// TIA Portal V18 export
FUNCTION_BLOCK "CentralShifter"   // FB10, LAD
{ S7_Optimized_Access := 'TRUE' }
// stored: MemoryReserve 100, SetENOAutomatically false
   VAR
      MC_POWER_CS_PP { S7_SetPoint := 'True'} : MC_POWER;
      MC_POWER_CS_PL { S7_SetPoint := 'True'} : MC_POWER;
      MC_POWER_CS_TP { S7_SetPoint := 'True'} : MC_POWER;
      MC_POWER_CS_TL { S7_SetPoint := 'True'} : MC_POWER;
      MC_POWER_CS_Virtual { S7_SetPoint := 'True'} : MC_POWER;
      MC_RESET_CS_PP { S7_SetPoint := 'True'} : MC_RESET;
      MC_RESET_CS_PL { S7_SetPoint := 'True'} : MC_RESET;
      MC_RESET_CS_TP { S7_SetPoint := 'True'} : MC_RESET;
      MC_RESET_CS_TL { S7_SetPoint := 'True'} : MC_RESET;
      MC_GEARIN_CS_PP { S7_SetPoint := 'True'} : MC_GEARIN;
      MC_GEARIN_CS_PL { S7_SetPoint := 'True'} : MC_GEARIN;
      MC_GEARIN_CS_TP { S7_SetPoint := 'True'} : MC_GEARIN;
      MC_GEARIN_CS_TL { S7_SetPoint := 'True'} : MC_GEARIN;
      MC_HOME_CS_PP { S7_SetPoint := 'True'} : MC_HOME;
      MC_HOME_CS_PL { S7_SetPoint := 'True'} : MC_HOME;
      MC_HOME_CS_TP { S7_SetPoint := 'True'} : MC_HOME;
      MC_HOME_CS_TL { S7_SetPoint := 'True'} : MC_HOME;
      MC_RESET_CS_Virtual { S7_SetPoint := 'True'} : MC_RESET;
      MC_MOVEJOG_CS_PL { S7_SetPoint := 'True'} : MC_MOVEJOG;
      MC_HOME_CS_Virtual { S7_SetPoint := 'True'} : MC_HOME;
      MC_MOVEJOG_CS_PP { S7_SetPoint := 'True'} : MC_MOVEJOG;
      MC_MOVEJOG_CS_TL { S7_SetPoint := 'True'} : MC_MOVEJOG;
      MC_MOVEJOG_CS_TP { S7_SetPoint := 'True'} : MC_MOVEJOG;
      MC_MOVEJOG_CS_Virtual { S7_SetPoint := 'True'} : MC_MOVEJOG;
      MC_MOVERELATIVE_CS_Virtual { S7_SetPoint := 'True'} : MC_MOVERELATIVE;
      MC_MOVEABSOLUTE_CS_Virtual { S7_SetPoint := 'True'} : MC_MOVEABSOLUTE;
      Homeing_Status { S7_SetPoint := 'True'} : Int;
      Jog_Backward_Home : Bool;
      Jog_Forward_Home : Bool;
      Jog_Velocity : Int;
   END_VAR
BEGIN

REGION Network 1
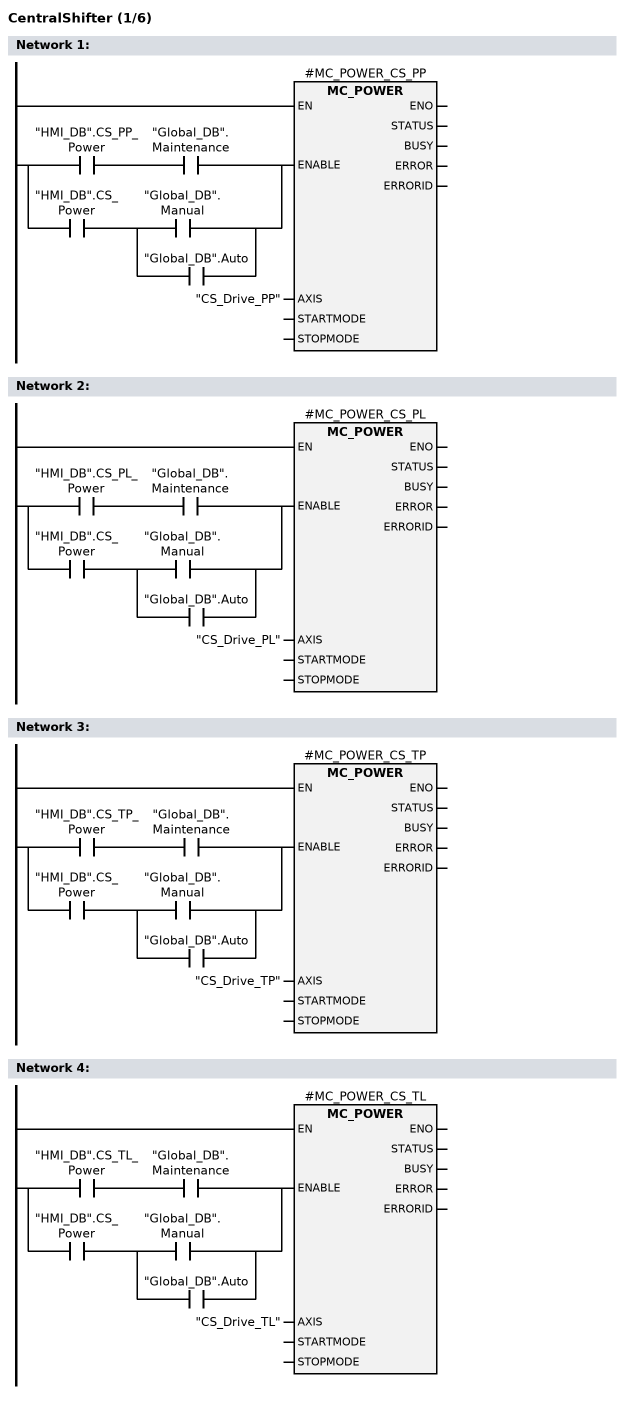
   RUNG wire#powerrail
      #MC_POWER_CS_PP.MC_POWER(Enable := wire#w2, Axis := "CS_Drive_PP", StartMode :=, StopMode :=, Status =>, Busy =>, Error =>, ErrorId =>)
   END_RUNG
   RUNG wire#powerrail
      Contact( "HMI_DB".CS_PP_Power )
      Contact( "Global_DB".Maintenance )
   END_RUNG wire#w2
   RUNG wire#powerrail
      Contact( "HMI_DB".CS_Power )
      wire#w1
      Contact( "Global_DB".Manual )
   END_RUNG wire#w2
   RUNG wire#w1
      Contact( "Global_DB".Auto )
   END_RUNG wire#w2
   // the same network as SCL:
   #MC_POWER_CS_PP(Enable := ("HMI_DB".CS_PP_Power AND "Global_DB".Maintenance) OR ("HMI_DB".CS_Power AND ("Global_DB".Manual OR "Global_DB".Auto)),   // MC_POWER
                   Axis := "CS_Drive_PP");
END_REGION

REGION Network 2
   RUNG wire#powerrail
      #MC_POWER_CS_PL.MC_POWER(Enable := wire#w2, Axis := "CS_Drive_PL", StartMode :=, StopMode :=, Status =>, Busy =>, Error =>, ErrorId =>)
   END_RUNG
   RUNG wire#powerrail
      Contact( "HMI_DB".CS_PL_Power )
      Contact( "Global_DB".Maintenance )
   END_RUNG wire#w2
   RUNG wire#powerrail
      Contact( "HMI_DB".CS_Power )
      wire#w1
      Contact( "Global_DB".Manual )
   END_RUNG wire#w2
   RUNG wire#w1
      Contact( "Global_DB".Auto )
   END_RUNG wire#w2
   // the same network as SCL:
   #MC_POWER_CS_PL(Enable := ("HMI_DB".CS_PL_Power AND "Global_DB".Maintenance) OR ("HMI_DB".CS_Power AND ("Global_DB".Manual OR "Global_DB".Auto)),   // MC_POWER
                   Axis := "CS_Drive_PL");
END_REGION

REGION Network 3
   RUNG wire#powerrail
      #MC_POWER_CS_TP.MC_POWER(Enable := wire#w2, Axis := "CS_Drive_TP", StartMode :=, StopMode :=, Status =>, Busy =>, Error =>, ErrorId =>)
   END_RUNG
   RUNG wire#powerrail
      Contact( "HMI_DB".CS_TP_Power )
      Contact( "Global_DB".Maintenance )
   END_RUNG wire#w2
   RUNG wire#powerrail
      Contact( "HMI_DB".CS_Power )
      wire#w1
      Contact( "Global_DB".Manual )
   END_RUNG wire#w2
   RUNG wire#w1
      Contact( "Global_DB".Auto )
   END_RUNG wire#w2
   // the same network as SCL:
   #MC_POWER_CS_TP(Enable := ("HMI_DB".CS_TP_Power AND "Global_DB".Maintenance) OR ("HMI_DB".CS_Power AND ("Global_DB".Manual OR "Global_DB".Auto)),   // MC_POWER
                   Axis := "CS_Drive_TP");
END_REGION

REGION Network 4
   RUNG wire#powerrail
      #MC_POWER_CS_TL.MC_POWER(Enable := wire#w2, Axis := "CS_Drive_TL", StartMode :=, StopMode :=, Status =>, Busy =>, Error =>, ErrorId =>)
   END_RUNG
   RUNG wire#powerrail
      Contact( "HMI_DB".CS_TL_Power )
      Contact( "Global_DB".Maintenance )
   END_RUNG wire#w2
   RUNG wire#powerrail
      Contact( "HMI_DB".CS_Power )
      wire#w1
      Contact( "Global_DB".Manual )
   END_RUNG wire#w2
   RUNG wire#w1
      Contact( "Global_DB".Auto )
   END_RUNG wire#w2
   // the same network as SCL:
   #MC_POWER_CS_TL(Enable := ("HMI_DB".CS_TL_Power AND "Global_DB".Maintenance) OR ("HMI_DB".CS_Power AND ("Global_DB".Manual OR "Global_DB".Auto)),   // MC_POWER
                   Axis := "CS_Drive_TL");
END_REGION

REGION Network 5
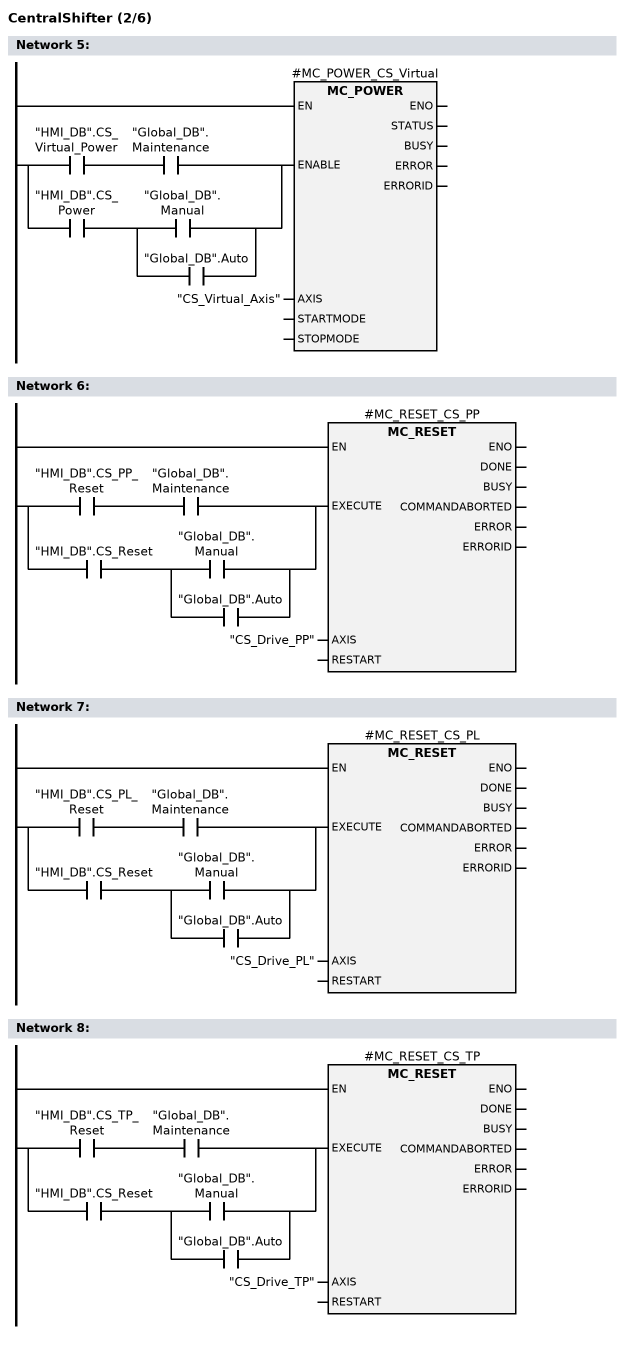
   RUNG wire#powerrail
      #MC_POWER_CS_Virtual.MC_POWER(Enable := wire#w2, Axis := "CS_Virtual_Axis", StartMode :=, StopMode :=, Status =>, Busy =>, Error =>, ErrorId =>)
   END_RUNG
   RUNG wire#powerrail
      Contact( "HMI_DB".CS_Virtual_Power )
      Contact( "Global_DB".Maintenance )
   END_RUNG wire#w2
   RUNG wire#powerrail
      Contact( "HMI_DB".CS_Power )
      wire#w1
      Contact( "Global_DB".Manual )
   END_RUNG wire#w2
   RUNG wire#w1
      Contact( "Global_DB".Auto )
   END_RUNG wire#w2
   // the same network as SCL:
   #MC_POWER_CS_Virtual(Enable := ("HMI_DB".CS_Virtual_Power AND "Global_DB".Maintenance) OR ("HMI_DB".CS_Power AND ("Global_DB".Manual OR "Global_DB".Auto)),   // MC_POWER
                        Axis := "CS_Virtual_Axis");
END_REGION

REGION Network 6
   RUNG wire#powerrail
      #MC_RESET_CS_PP.MC_RESET(Execute := wire#w2, Axis := "CS_Drive_PP", Restart :=, Done =>, Busy =>, CommandAborted =>, Error =>, ErrorId =>)
   END_RUNG
   RUNG wire#powerrail
      Contact( "HMI_DB".CS_PP_Reset )
      Contact( "Global_DB".Maintenance )
   END_RUNG wire#w2
   RUNG wire#powerrail
      Contact( "HMI_DB".CS_Reset )
      wire#w1
      Contact( "Global_DB".Manual )
   END_RUNG wire#w2
   RUNG wire#w1
      Contact( "Global_DB".Auto )
   END_RUNG wire#w2
   // the same network as SCL:
   #MC_RESET_CS_PP(Execute := ("HMI_DB".CS_PP_Reset AND "Global_DB".Maintenance) OR ("HMI_DB".CS_Reset AND ("Global_DB".Manual OR "Global_DB".Auto)),   // MC_RESET
                   Axis := "CS_Drive_PP");
END_REGION

REGION Network 7
   RUNG wire#powerrail
      #MC_RESET_CS_PL.MC_RESET(Execute := wire#w2, Axis := "CS_Drive_PL", Restart :=, Done =>, Busy =>, CommandAborted =>, Error =>, ErrorId =>)
   END_RUNG
   RUNG wire#powerrail
      Contact( "HMI_DB".CS_PL_Reset )
      Contact( "Global_DB".Maintenance )
   END_RUNG wire#w2
   RUNG wire#powerrail
      Contact( "HMI_DB".CS_Reset )
      wire#w1
      Contact( "Global_DB".Manual )
   END_RUNG wire#w2
   RUNG wire#w1
      Contact( "Global_DB".Auto )
   END_RUNG wire#w2
   // the same network as SCL:
   #MC_RESET_CS_PL(Execute := ("HMI_DB".CS_PL_Reset AND "Global_DB".Maintenance) OR ("HMI_DB".CS_Reset AND ("Global_DB".Manual OR "Global_DB".Auto)),   // MC_RESET
                   Axis := "CS_Drive_PL");
END_REGION

REGION Network 8
   RUNG wire#powerrail
      #MC_RESET_CS_TP.MC_RESET(Execute := wire#w2, Axis := "CS_Drive_TP", Restart :=, Done =>, Busy =>, CommandAborted =>, Error =>, ErrorId =>)
   END_RUNG
   RUNG wire#powerrail
      Contact( "HMI_DB".CS_TP_Reset )
      Contact( "Global_DB".Maintenance )
   END_RUNG wire#w2
   RUNG wire#powerrail
      Contact( "HMI_DB".CS_Reset )
      wire#w1
      Contact( "Global_DB".Manual )
   END_RUNG wire#w2
   RUNG wire#w1
      Contact( "Global_DB".Auto )
   END_RUNG wire#w2
   // the same network as SCL:
   #MC_RESET_CS_TP(Execute := ("HMI_DB".CS_TP_Reset AND "Global_DB".Maintenance) OR ("HMI_DB".CS_Reset AND ("Global_DB".Manual OR "Global_DB".Auto)),   // MC_RESET
                   Axis := "CS_Drive_TP");
END_REGION

REGION Network 9
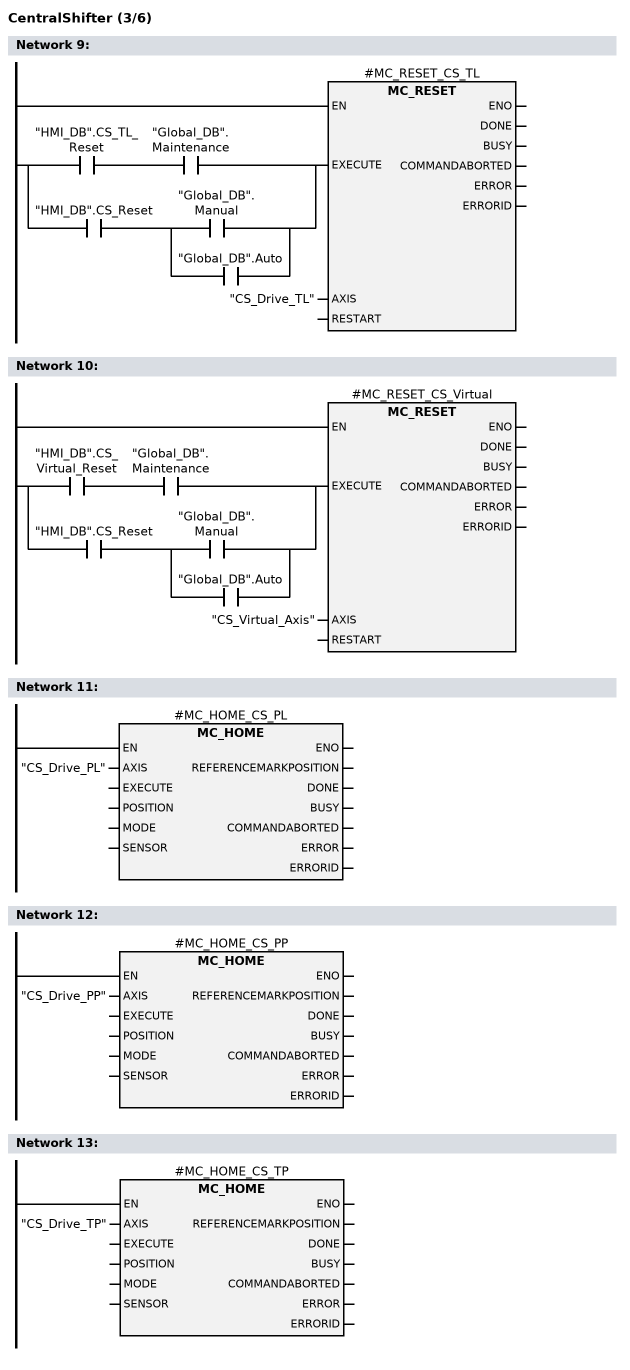
   RUNG wire#powerrail
      #MC_RESET_CS_TL.MC_RESET(Execute := wire#w2, Axis := "CS_Drive_TL", Restart :=, Done =>, Busy =>, CommandAborted =>, Error =>, ErrorId =>)
   END_RUNG
   RUNG wire#powerrail
      Contact( "HMI_DB".CS_TL_Reset )
      Contact( "Global_DB".Maintenance )
   END_RUNG wire#w2
   RUNG wire#powerrail
      Contact( "HMI_DB".CS_Reset )
      wire#w1
      Contact( "Global_DB".Manual )
   END_RUNG wire#w2
   RUNG wire#w1
      Contact( "Global_DB".Auto )
   END_RUNG wire#w2
   // the same network as SCL:
   #MC_RESET_CS_TL(Execute := ("HMI_DB".CS_TL_Reset AND "Global_DB".Maintenance) OR ("HMI_DB".CS_Reset AND ("Global_DB".Manual OR "Global_DB".Auto)),   // MC_RESET
                   Axis := "CS_Drive_TL");
END_REGION

REGION Network 10
   RUNG wire#powerrail
      #MC_RESET_CS_Virtual.MC_RESET(Execute := wire#w2, Axis := "CS_Virtual_Axis", Restart :=, Done =>, Busy =>, CommandAborted =>, Error =>, ErrorId =>)
   END_RUNG
   RUNG wire#powerrail
      Contact( "HMI_DB".CS_Virtual_Reset )
      Contact( "Global_DB".Maintenance )
   END_RUNG wire#w2
   RUNG wire#powerrail
      Contact( "HMI_DB".CS_Reset )
      wire#w1
      Contact( "Global_DB".Manual )
   END_RUNG wire#w2
   RUNG wire#w1
      Contact( "Global_DB".Auto )
   END_RUNG wire#w2
   // the same network as SCL:
   #MC_RESET_CS_Virtual(Execute := ("HMI_DB".CS_Virtual_Reset AND "Global_DB".Maintenance) OR ("HMI_DB".CS_Reset AND ("Global_DB".Manual OR "Global_DB".Auto)),   // MC_RESET
                        Axis := "CS_Virtual_Axis");
END_REGION

REGION Network 11
   RUNG wire#powerrail
      #MC_HOME_CS_PL.MC_HOME(Axis := "CS_Drive_PL", Execute :=, Position :=, Mode :=, Sensor :=, ReferenceMarkPosition =>, Done =>, Busy =>, CommandAborted =>, Error =>, ErrorId =>)
   END_RUNG
   // the same network as SCL:
   #MC_HOME_CS_PL(Axis := "CS_Drive_PL");   // MC_HOME
END_REGION

REGION Network 12
   RUNG wire#powerrail
      #MC_HOME_CS_PP.MC_HOME(Axis := "CS_Drive_PP", Execute :=, Position :=, Mode :=, Sensor :=, ReferenceMarkPosition =>, Done =>, Busy =>, CommandAborted =>, Error =>, ErrorId =>)
   END_RUNG
   // the same network as SCL:
   #MC_HOME_CS_PP(Axis := "CS_Drive_PP");   // MC_HOME
END_REGION

REGION Network 13
   RUNG wire#powerrail
      #MC_HOME_CS_TP.MC_HOME(Axis := "CS_Drive_TP", Execute :=, Position :=, Mode :=, Sensor :=, ReferenceMarkPosition =>, Done =>, Busy =>, CommandAborted =>, Error =>, ErrorId =>)
   END_RUNG
   // the same network as SCL:
   #MC_HOME_CS_TP(Axis := "CS_Drive_TP");   // MC_HOME
END_REGION

REGION Network 14
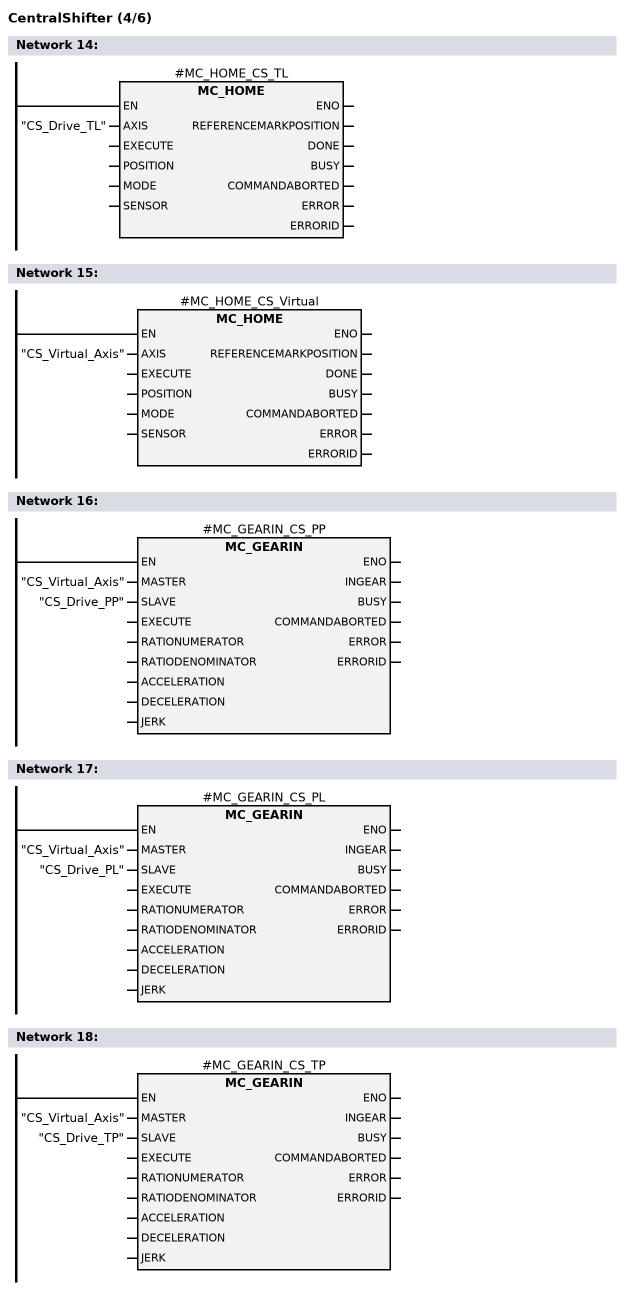
   RUNG wire#powerrail
      #MC_HOME_CS_TL.MC_HOME(Axis := "CS_Drive_TL", Execute :=, Position :=, Mode :=, Sensor :=, ReferenceMarkPosition =>, Done =>, Busy =>, CommandAborted =>, Error =>, ErrorId =>)
   END_RUNG
   // the same network as SCL:
   #MC_HOME_CS_TL(Axis := "CS_Drive_TL");   // MC_HOME
END_REGION

REGION Network 15
   RUNG wire#powerrail
      #MC_HOME_CS_Virtual.MC_HOME(Axis := "CS_Virtual_Axis", Execute :=, Position :=, Mode :=, Sensor :=, ReferenceMarkPosition =>, Done =>, Busy =>, CommandAborted =>, Error =>, ErrorId =>)
   END_RUNG
   // the same network as SCL:
   #MC_HOME_CS_Virtual(Axis := "CS_Virtual_Axis");   // MC_HOME
END_REGION

REGION Network 16
   RUNG wire#powerrail
      #MC_GEARIN_CS_PP.MC_GEARIN(Master := "CS_Virtual_Axis", Slave := "CS_Drive_PP", Execute :=, RatioNumerator :=, RatioDenominator :=, Acceleration :=, Deceleration :=, Jerk :=, InGear =>, Busy =>, CommandAborted =>, Error =>, ErrorId =>)
   END_RUNG
   // the same network as SCL:
   #MC_GEARIN_CS_PP(Master := "CS_Virtual_Axis", Slave := "CS_Drive_PP");   // MC_GEARIN
END_REGION

REGION Network 17
   RUNG wire#powerrail
      #MC_GEARIN_CS_PL.MC_GEARIN(Master := "CS_Virtual_Axis", Slave := "CS_Drive_PL", Execute :=, RatioNumerator :=, RatioDenominator :=, Acceleration :=, Deceleration :=, Jerk :=, InGear =>, Busy =>, CommandAborted =>, Error =>, ErrorId =>)
   END_RUNG
   // the same network as SCL:
   #MC_GEARIN_CS_PL(Master := "CS_Virtual_Axis", Slave := "CS_Drive_PL");   // MC_GEARIN
END_REGION

REGION Network 18
   RUNG wire#powerrail
      #MC_GEARIN_CS_TP.MC_GEARIN(Master := "CS_Virtual_Axis", Slave := "CS_Drive_TP", Execute :=, RatioNumerator :=, RatioDenominator :=, Acceleration :=, Deceleration :=, Jerk :=, InGear =>, Busy =>, CommandAborted =>, Error =>, ErrorId =>)
   END_RUNG
   // the same network as SCL:
   #MC_GEARIN_CS_TP(Master := "CS_Virtual_Axis", Slave := "CS_Drive_TP");   // MC_GEARIN
END_REGION

REGION Network 19
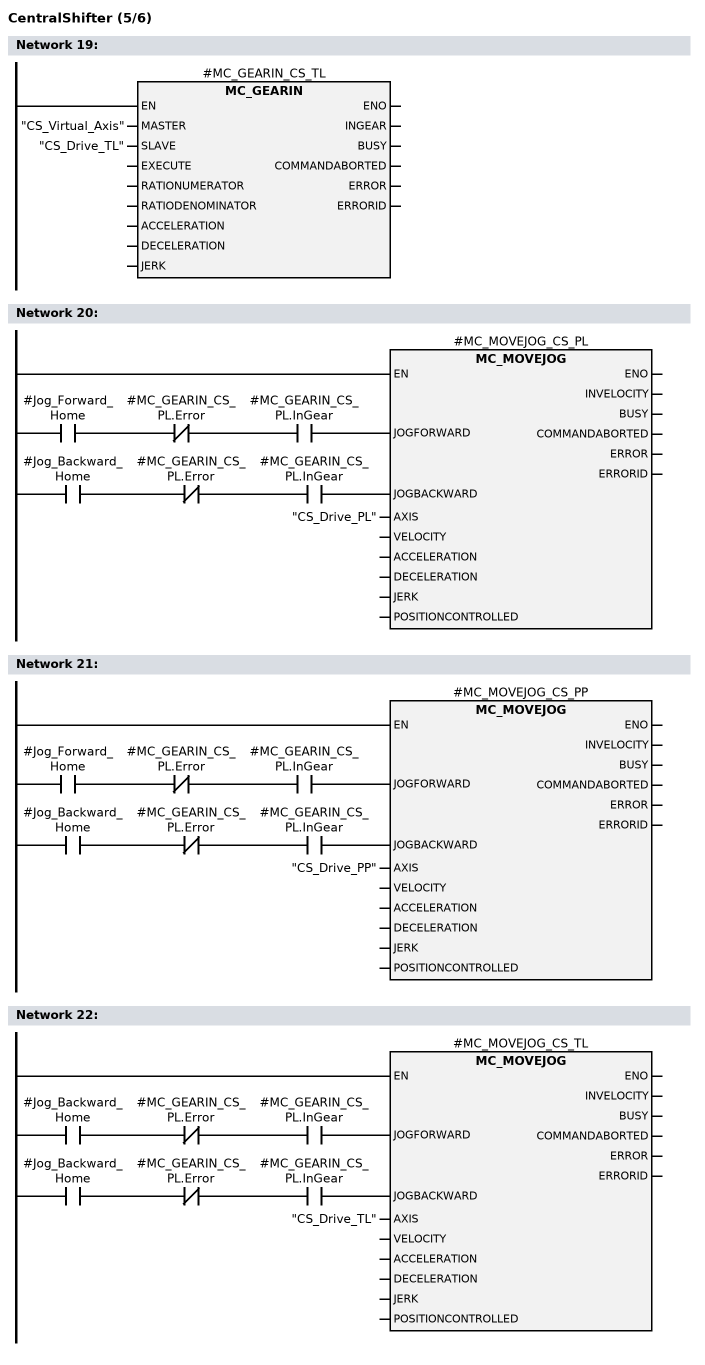
   RUNG wire#powerrail
      #MC_GEARIN_CS_TL.MC_GEARIN(Master := "CS_Virtual_Axis", Slave := "CS_Drive_TL", Execute :=, RatioNumerator :=, RatioDenominator :=, Acceleration :=, Deceleration :=, Jerk :=, InGear =>, Busy =>, CommandAborted =>, Error =>, ErrorId =>)
   END_RUNG
   // the same network as SCL:
   #MC_GEARIN_CS_TL(Master := "CS_Virtual_Axis", Slave := "CS_Drive_TL");   // MC_GEARIN
END_REGION

REGION Network 20
   RUNG wire#powerrail
      #MC_MOVEJOG_CS_PL.MC_MOVEJOG(JogForward := wire#w1, JogBackward := wire#w2, Axis := "CS_Drive_PL", Velocity :=, Acceleration :=, Deceleration :=, Jerk :=, PositionControlled :=, InVelocity =>, Busy =>, CommandAborted =>, Error =>, ErrorId =>)
   END_RUNG
   RUNG wire#powerrail
      Contact( #Jog_Forward_Home )
      I_Contact( #MC_GEARIN_CS_PL.Error )
      Contact( #MC_GEARIN_CS_PL.InGear )
   END_RUNG wire#w1
   RUNG wire#powerrail
      Contact( #Jog_Backward_Home )
      I_Contact( #MC_GEARIN_CS_PL.Error )
      Contact( #MC_GEARIN_CS_PL.InGear )
   END_RUNG wire#w2
   // the same network as SCL:
   #MC_MOVEJOG_CS_PL(JogForward := #Jog_Forward_Home AND NOT #MC_GEARIN_CS_PL.Error AND #MC_GEARIN_CS_PL.InGear,   // MC_MOVEJOG
                     JogBackward := #Jog_Backward_Home AND NOT #MC_GEARIN_CS_PL.Error AND #MC_GEARIN_CS_PL.InGear,
                     Axis := "CS_Drive_PL");
END_REGION

REGION Network 21
   RUNG wire#powerrail
      #MC_MOVEJOG_CS_PP.MC_MOVEJOG(JogForward := wire#w1, JogBackward := wire#w2, Axis := "CS_Drive_PP", Velocity :=, Acceleration :=, Deceleration :=, Jerk :=, PositionControlled :=, InVelocity =>, Busy =>, CommandAborted =>, Error =>, ErrorId =>)
   END_RUNG
   RUNG wire#powerrail
      Contact( #Jog_Forward_Home )
      I_Contact( #MC_GEARIN_CS_PL.Error )
      Contact( #MC_GEARIN_CS_PL.InGear )
   END_RUNG wire#w1
   RUNG wire#powerrail
      Contact( #Jog_Backward_Home )
      I_Contact( #MC_GEARIN_CS_PL.Error )
      Contact( #MC_GEARIN_CS_PL.InGear )
   END_RUNG wire#w2
   // the same network as SCL:
   #MC_MOVEJOG_CS_PP(JogForward := #Jog_Forward_Home AND NOT #MC_GEARIN_CS_PL.Error AND #MC_GEARIN_CS_PL.InGear,   // MC_MOVEJOG
                     JogBackward := #Jog_Backward_Home AND NOT #MC_GEARIN_CS_PL.Error AND #MC_GEARIN_CS_PL.InGear,
                     Axis := "CS_Drive_PP");
END_REGION

REGION Network 22
   RUNG wire#powerrail
      #MC_MOVEJOG_CS_TL.MC_MOVEJOG(JogForward := wire#w1, JogBackward := wire#w2, Axis := "CS_Drive_TL", Velocity :=, Acceleration :=, Deceleration :=, Jerk :=, PositionControlled :=, InVelocity =>, Busy =>, CommandAborted =>, Error =>, ErrorId =>)
   END_RUNG
   RUNG wire#powerrail
      Contact( #Jog_Backward_Home )
      I_Contact( #MC_GEARIN_CS_PL.Error )
      Contact( #MC_GEARIN_CS_PL.InGear )
   END_RUNG wire#w1
   RUNG wire#powerrail
      Contact( #Jog_Backward_Home )
      I_Contact( #MC_GEARIN_CS_PL.Error )
      Contact( #MC_GEARIN_CS_PL.InGear )
   END_RUNG wire#w2
   // the same network as SCL:
   #MC_MOVEJOG_CS_TL(JogForward := #Jog_Backward_Home AND NOT #MC_GEARIN_CS_PL.Error AND #MC_GEARIN_CS_PL.InGear,   // MC_MOVEJOG
                     JogBackward := #Jog_Backward_Home AND NOT #MC_GEARIN_CS_PL.Error AND #MC_GEARIN_CS_PL.InGear,
                     Axis := "CS_Drive_TL");
END_REGION

REGION Network 23
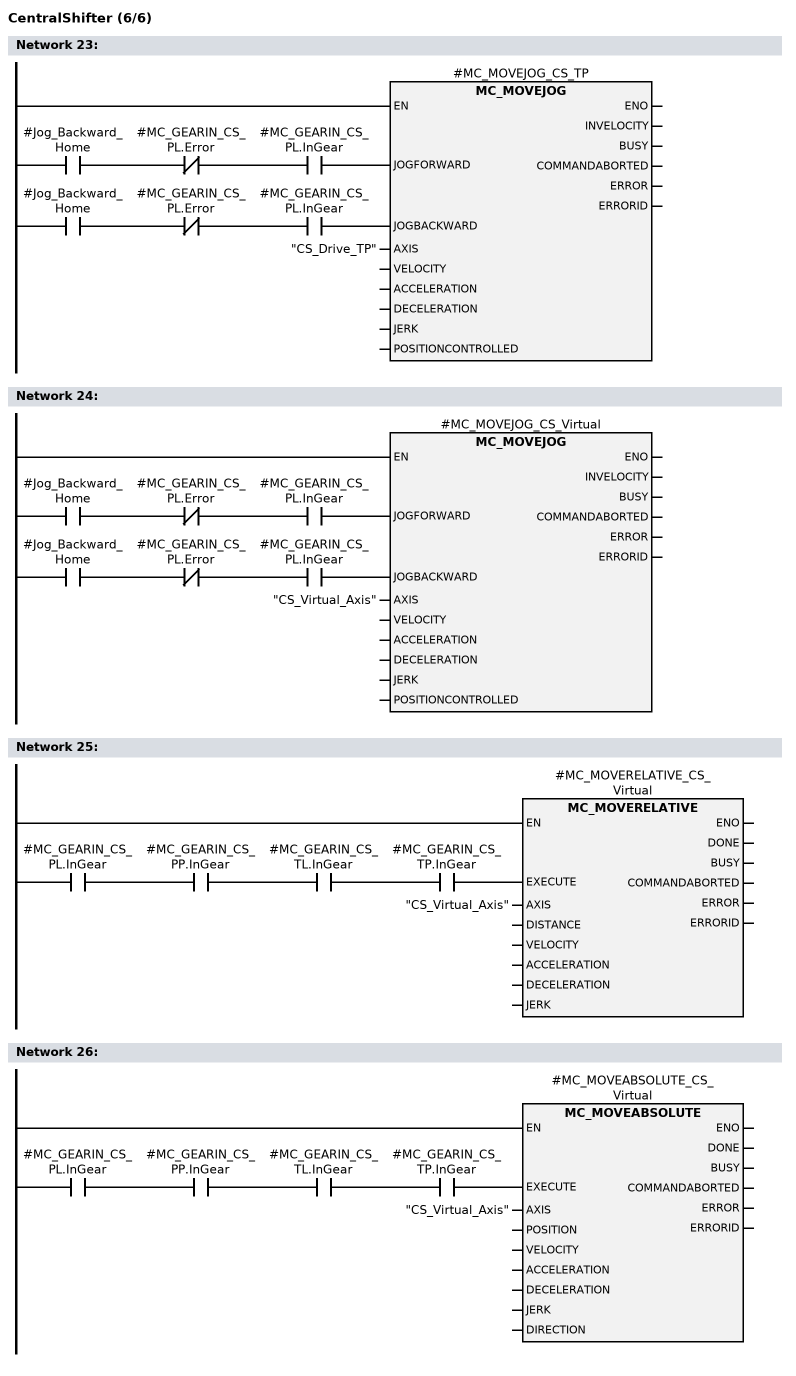
   RUNG wire#powerrail
      #MC_MOVEJOG_CS_TP.MC_MOVEJOG(JogForward := wire#w1, JogBackward := wire#w2, Axis := "CS_Drive_TP", Velocity :=, Acceleration :=, Deceleration :=, Jerk :=, PositionControlled :=, InVelocity =>, Busy =>, CommandAborted =>, Error =>, ErrorId =>)
   END_RUNG
   RUNG wire#powerrail
      Contact( #Jog_Backward_Home )
      I_Contact( #MC_GEARIN_CS_PL.Error )
      Contact( #MC_GEARIN_CS_PL.InGear )
   END_RUNG wire#w1
   RUNG wire#powerrail
      Contact( #Jog_Backward_Home )
      I_Contact( #MC_GEARIN_CS_PL.Error )
      Contact( #MC_GEARIN_CS_PL.InGear )
   END_RUNG wire#w2
   // the same network as SCL:
   #MC_MOVEJOG_CS_TP(JogForward := #Jog_Backward_Home AND NOT #MC_GEARIN_CS_PL.Error AND #MC_GEARIN_CS_PL.InGear,   // MC_MOVEJOG
                     JogBackward := #Jog_Backward_Home AND NOT #MC_GEARIN_CS_PL.Error AND #MC_GEARIN_CS_PL.InGear,
                     Axis := "CS_Drive_TP");
END_REGION

REGION Network 24
   RUNG wire#powerrail
      #MC_MOVEJOG_CS_Virtual.MC_MOVEJOG(JogForward := wire#w1, JogBackward := wire#w2, Axis := "CS_Virtual_Axis", Velocity :=, Acceleration :=, Deceleration :=, Jerk :=, PositionControlled :=, InVelocity =>, Busy =>, CommandAborted =>, Error =>, ErrorId =>)
   END_RUNG
   RUNG wire#powerrail
      Contact( #Jog_Backward_Home )
      I_Contact( #MC_GEARIN_CS_PL.Error )
      Contact( #MC_GEARIN_CS_PL.InGear )
   END_RUNG wire#w1
   RUNG wire#powerrail
      Contact( #Jog_Backward_Home )
      I_Contact( #MC_GEARIN_CS_PL.Error )
      Contact( #MC_GEARIN_CS_PL.InGear )
   END_RUNG wire#w2
   // the same network as SCL:
   #MC_MOVEJOG_CS_Virtual(JogForward := #Jog_Backward_Home AND NOT #MC_GEARIN_CS_PL.Error AND #MC_GEARIN_CS_PL.InGear,   // MC_MOVEJOG
                          JogBackward := #Jog_Backward_Home AND NOT #MC_GEARIN_CS_PL.Error AND #MC_GEARIN_CS_PL.InGear,
                          Axis := "CS_Virtual_Axis");
END_REGION

REGION Network 25
   RUNG wire#powerrail
      #MC_MOVERELATIVE_CS_Virtual.MC_MOVERELATIVE(Execute := wire#w1, Axis := "CS_Virtual_Axis", Distance :=, Velocity :=, Acceleration :=, Deceleration :=, Jerk :=, Done =>, Busy =>, CommandAborted =>, Error =>, ErrorId =>)
   END_RUNG
   RUNG wire#powerrail
      Contact( #MC_GEARIN_CS_PL.InGear )
      Contact( #MC_GEARIN_CS_PP.InGear )
      Contact( #MC_GEARIN_CS_TL.InGear )
      Contact( #MC_GEARIN_CS_TP.InGear )
   END_RUNG wire#w1
   // the same network as SCL:
   #MC_MOVERELATIVE_CS_Virtual(Execute := #MC_GEARIN_CS_PL.InGear AND #MC_GEARIN_CS_PP.InGear AND #MC_GEARIN_CS_TL.InGear AND #MC_GEARIN_CS_TP.InGear,   // MC_MOVERELATIVE
                           Axis := "CS_Virtual_Axis");
END_REGION

REGION Network 26
   RUNG wire#powerrail
      #MC_MOVEABSOLUTE_CS_Virtual.MC_MOVEABSOLUTE(Execute := wire#w1, Axis := "CS_Virtual_Axis", Position :=, Velocity :=, Acceleration :=, Deceleration :=, Jerk :=, Direction :=, Done =>, Busy =>, CommandAborted =>, Error =>, ErrorId =>)
   END_RUNG
   RUNG wire#powerrail
      Contact( #MC_GEARIN_CS_PL.InGear )
      Contact( #MC_GEARIN_CS_PP.InGear )
      Contact( #MC_GEARIN_CS_TL.InGear )
      Contact( #MC_GEARIN_CS_TP.InGear )
   END_RUNG wire#w1
   // the same network as SCL:
   #MC_MOVEABSOLUTE_CS_Virtual(Execute := #MC_GEARIN_CS_PL.InGear AND #MC_GEARIN_CS_PP.InGear AND #MC_GEARIN_CS_TL.InGear AND #MC_GEARIN_CS_TP.InGear,   // MC_MOVEABSOLUTE
                           Axis := "CS_Virtual_Axis");
END_REGION

REGION Network 27 (SCL): Homing
   IF "HMI_DB".CS_Homing AND NOT "iCS_SensorHoming_Left" AND (#Homeing_Status = 0 OR #Homeing_Status = 5) THEN
       #Jog_Backward_Home := 1;
       #Jog_Forward_Home := 0;
       #Jog_Velocity := 15;
       #Homeing_Status := 1;

   ELSIF "HMI_DB".CS_Homing  AND "iCS_SensorHoming_Left" THEN
       #Jog_Backward_Home := 0;
       #Jog_Forward_Home := 1;
       #Jog_Velocity := 1;
       #Homeing_Status := 2;

   ELSIF "HMI_DB".CS_Homing  AND NOT "iCS_SensorHoming_Left" AND #Homeing_Status = 2 THEN
       #Jog_Backward_Home := 0;
       #Jog_Forward_Home := 0;
       #Homeing_Status := 3;

   ELSIF "HMI_DB".CS_Homing AND NOT "iCS_SensorHoming_Left" AND #Homeing_Status = 3 THEN
       #MC_HOME_CS_PL.Execute := 1;
       #MC_HOME_CS_PP.Execute := 1;
       #MC_HOME_CS_TP.Execute := 1;
       #MC_HOME_CS_TL.Execute := 1;
       #MC_HOME_CS_Virtual.Execute := 1;
       #Homeing_Status := 4;
       "HMI_DB".CS_Homing := 0;

   ELSIF #Homeing_Status = 4 AND #MC_HOME_CS_PL.Done AND #MC_HOME_CS_PL.Done AND #MC_HOME_CS_TL.Done AND #MC_HOME_CS_TL.Done AND #MC_HOME_CS_Virtual.Done AND "CS_Virtual_Axis".Position <= 1 THEN
       #MC_HOME_CS_PL.Execute := 0;
       #MC_HOME_CS_PP.Execute := 0;
       #MC_HOME_CS_TP.Execute := 0;
       #MC_HOME_CS_TL.Execute := 0;
       #Homeing_Status := 5; //ready
       "HMI_DB".CS_Homing := 0;

   ELSIF #Homeing_Status = 5 THEN
       "HMI_DB".CS_Homing := 0;
       IF "CS_Virtual_Axis".Position >= 1 THEN
           #Homeing_Status := 0;

       END_IF;
   END_IF;
END_REGION
END_FUNCTION_BLOCK
